//HERE  YOU CAN WRITE  WHAT IS NECESSARY 
//TO SUPSEND  PROCESS..... TO INTERUPT SAFETY

IF (Step(1000, TRUE, '<#SUSPENDING COMPONENTS#>')) THEN
 	//-------------------------------------    
	//StepCompleteWhen(Station.AutomatTask.CurrentStep.Status <> eStepStatus.Running);
		
    StepCompleteWhen( CurrentStep.Duration >= T#3000MS);
    //-------------------------------------
END_IF

IF (Step(30000, TRUE, 'SUSPEND DONE')) THEN
    //-------------------------------------
		
        THIS^._done:=TRUE;
		THIS^.Task.DoneWhen(TRUE);
	
   
    //-------------------------------------	
END_IF
END_METHOD

METHOD PUBLIC OnStart
SUPER^.OnStart();
Station.RecoverTask.Restore();
END_METHOD

PROPERTY Station : REFERENCE TO CU00x
GET
VAR
    _station : POINTER TO CU00x;
END_VAR
IF __QUERYPOINTER(Parent, _station) THEN // Check if _Parent is Station001
    Station REF= _station^;              // If the check is successful dereference a pointer. simlar to THIS^ or SUPER^
END_IF
END_GET
END_PROPERTY

END_FUNCTION_BLOCK

// ---- Abstractions/CUBase/Tasks/CUBaseSuspend.TcPOU
FUNCTION_BLOCK ABSTRACT CUBaseSuspend EXTENDS TcoTaskedSequencer
VAR
	_done:BOOL;

END_VAR

PROPERTY Done : bool
GET
Done := _done;
END_GET
END_PROPERTY

METHOD PUBLIC OnStart
_done:=FALSE;
END_METHOD

PROPERTY StationBase : REFERENCE TO CuBase
GET
VAR
    _station : POINTER TO CuBase;
END_VAR
IF __QUERYPOINTER(Parent, _station) THEN // Check if _Parent is Station001
    StationBase REF= _station^;              // If the check is successful dereference a pointer. simlar to THIS^ or SUPER^
END_IF
END_GET
END_PROPERTY

END_FUNCTION_BLOCK

// ---- Technology/CU00x/Safety/Recover/CU00xRecoverTask.TcPOU
FUNCTION_BLOCK CU00xRecoverTask EXTENDS CUBaseRecover IMPLEMENTS ICUTask
VAR
	_sb : TcoCore.StringBuilder;
END_VAR

Run();

(*~
	<docu>
		<summary>
			Main method of the sequener. Custom code needs to be placed here. The sequencer is executed by call of **Instance.Run()** method.
			This method is abstract, and it must be overridden in derived block.
		</summary>
	</docu>
~*)
METHOD PROTECTED Main : BOOL
(*

	RECOVER PROCESS 
	Following steps provide recover action for this controlled unit.
	Add components add write customized sequence according to your need.
*)

		
//
IF (Step(100, TRUE, '<#WAITING FOR START#>')) THEN
    //-------------------------------------    

    StepCompleteWhen(TRUE);
    //-------------------------------------
END_IF

//HERE  YOU CAN WRITE  WHAT IS NECESSARY 
//TO RECOVER AFTER INTERUPTED PROCESS.....

IF (Step(1000, TRUE, '<#RECOVER ANY COMPONENTS#>')) THEN
    //-------------------------------------    

    StepCompleteWhen(CurrentStep.Duration >= T#3000MS);
    //-------------------------------------
END_IF

IF (Step(30000, TRUE, 'RECOVER DONE')) THEN
    //-------------------------------------
		
        this^._done:=true;
		THIS^.Task.DoneWhen(TRUE);
		
   
    //-------------------------------------	
END_IF
END_METHOD

METHOD PUBLIC OnStart
SUPER^.OnStart();
Station.SuspendTask.Restore();
END_METHOD

PROPERTY Station : REFERENCE TO CU00x
GET
VAR
    _station : POINTER TO CU00x;
END_VAR
IF __QUERYPOINTER(Parent, _station) THEN // Check if _Parent is Station001
    Station REF= _station^;              // If the check is successful dereference a pointer. simlar to THIS^ or SUPER^
END_IF
END_GET
END_PROPERTY

END_FUNCTION_BLOCK

// ---- Abstractions/CUBase/Tasks/CUBaseRecover.TcPOU
FUNCTION_BLOCK ABSTRACT CUBaseRecover EXTENDS TcoTaskedSequencer
VAR
	_done:BOOL;

END_VAR

PROPERTY Done : bool
GET
Done := _done;
END_GET
END_PROPERTY

METHOD PUBLIC OnStart
_done:=FALSE;
END_METHOD

PROPERTY StationBase : REFERENCE TO CuBase
GET
VAR
    _station : POINTER TO CuBase;
END_VAR
IF __QUERYPOINTER(Parent, _station) THEN // Check if _Parent is Station001
    StationBase REF= _station^;              // If the check is successful dereference a pointer. simlar to THIS^ or SUPER^
END_IF
END_GET
END_PROPERTY

END_FUNCTION_BLOCK

// ---- Technology/CU00x/Positions/Cu00xTestPositions.TcPOU
FUNCTION_BLOCK Cu00xTestPositions EXTENDS TcoDrivesBeckhoff.TcoSingleAxisPositionsRootContainer
VAR_INPUT
END_VAR
VAR_OUTPUT
END_VAR
VAR
	{attribute addProperty Name "<#Pick Position#>"}
	PickPosition:TcoDrivesBeckhoff.TcoSingleAxisMoveParam;
	{attribute addProperty Name "<#Place  Position#>"}
	PlacePosition:TcoDrivesBeckhoff.TcoSingleAxisMoveParam;
END_VAR

END_FUNCTION_BLOCK

// ---- Technology/CU00x/Positions/CU00xTestMultiPositions.TcPOU
FUNCTION_BLOCK CU00xTestMultiPositions EXTENDS TcoDrivesBeckhoff.TcoMultiAxisPositionsRootContainer
VAR_INPUT
END_VAR
VAR_OUTPUT
END_VAR
VAR
	{attribute addProperty Name "<#Pick Position#>"}
	PickPosition:TcoDrivesBeckhoff.TcoMultiAxisMoveParam;
	{attribute addProperty Name "<#Place  Position#>"}
	PlacePosition:TcoDrivesBeckhoff.TcoMultiAxisMoveParam;

END_VAR

PROPERTY PUBLIC PickPos : REFERENCE TO TcoDrivesBeckhoff.TcoMultiAxisMoveParam;
GET
PickPos REF=PickPosition;
END_GET
END_PROPERTY

PROPERTY PUBLIC PlacePos : REFERENCE TO TcoDrivesBeckhoff.TcoMultiAxisMoveParam;
GET
PlacePos REF=PlacePosition;
END_GET
END_PROPERTY

END_FUNCTION_BLOCK

// ---- Abstractions/Generic/LightTower/TcoLightTower.TcPOU
FUNCTION_BLOCK TcoLightTower EXTENDS TcoCore.TcoComponent
VAR_IN_OUT
	{attribute clr [RenderIgnore()]}
	inoGreenLight   :  BOOL;
	
	{attribute clr [RenderIgnore()]}
	inoRedLight     :  BOOL;
	
	{attribute clr [RenderIgnore()]}
	inoOrangeLight  :  BOOL;
	
	{attribute clr [RenderIgnore()]}
	inoBlueLight    :  BOOL;

	{attribute clr [RenderIgnore()]}
	inoHorn         :  BOOL;
END_VAR

VAR
	
	
	{attribute addProperty Name "<#Status#>"}
    {attribute clr [ReadOnly()]}
    _status : TcoLightTower_Status;

	{attribute addProperty Name "<#Config#>"}
    _config : TcoLightTower_Config;
	
    _materrialError : bool;

	{attribute clr [RenderIgnore()]}
	_controlledUnits      : ARRAY [0..12] OF ICUBase;
				
	
	
	// group states

	{attribute clr [RenderIgnore()]}
	_blinker              : TcoUtilities.TcoBlinker(THIS^);
	{attribute clr [RenderIgnore()]}
	_blinkerSlow              : TcoUtilities.TcoBlinker(THIS^);
	

END_VAR

IF _controlledUnits[0] = 0 THEN
    THIS^.Messenger.Programming('<#Missing link to Controlled unit! No function is being executed!#>');
    RETURN;
END_IF

inoGreenLight := FALSE;
inoRedLight := FALSE;
inoOrangeLight := FALSE;
inoBlueLight := FALSE;
inoHorn := FALSE;

_blinker(inOffTime := T#500MS, inOnTime := T#500MS); //2 Hz
_blinkerSlow(inOffTime := T#1250MS, inOnTime := T#1250MS); //0.8 Hz

THIS^.Initialize();

//ground
IF _status.State.AnyGrounding THEN
    inoGreenLight := _blinker.IsOn;
    inoRedLight := _status.State.AnyInError AND _blinker.IsOn;
    inoOrangeLight := _status.State.AnyInWarning AND _blinker.IsOn;
END_IF

//auto
IF _status.State.AllInAuto AND NOT _status.State.AnyInStepMode AND NOT _status.State.AnyInError AND _status.State.AnyInWarning THEN
    inoGreenLight := TRUE; // ok production
ELSIF _status.State.AllInAuto AND _status.State.AnyInStepMode THEN
    inoGreenLight := _blinker.IsOn; //step mode
ELSIF _status.State.AllInAuto AND NOT _status.State.AnyInStepMode THEN
    inoGreenLight := TRUE; // ok production
    inoRedLight := _status.State.AnyInError AND _blinker.IsOn;
    inoOrangeLight := _status.State.AnyInWarning AND _blinker.IsOn;
ELSIF _status.State.AllInManual  THEN

    inoOrangeLight :=  _blinker.IsOn;

END_IF;

IF NOT _config.HornEnabled THEN
    inoHorn := FALSE;
END_IF;

//todo blue should be suitable for material feeding
IF _materrialError AND _status.State.AllInAuto THEN
	inoBlueLight :=  _blinker.IsOn;
END_IF

METHOD AddControlledUnit : BOOL
VAR_INPUT
 	inControlledUnit : ICUBase;
END_VAR
VAR
	i : UINT;
END_VAR
AddControlledUnit := FALSE;

IF inControlledUnit = 0 THEN
	RETURN;
END_IF

FOR i := 0 TO _config.MaxControledUnits DO
	IF _controlledUnits[i] = inControlledUnit THEN
		AddControlledUnit := TRUE;
		RETURN;
	END_IF
	
	IF 	_controlledUnits[i] = 0 THEN
		_controlledUnits[i] := inControlledUnit;
		AddControlledUnit    := TRUE;
		RETURN;
	END_IF
END_FOR
END_METHOD

PROPERTY Config :REFERENCE TO TcoLightTower_Config
GET
Config ref=_config;
END_GET
END_PROPERTY

METHOD Initialize : BOOL
VAR
	i : UINT;

END_VAR
_status.State.AllInAuto := TRUE;
_status.State.AllInGrounding := TRUE;
_status.State.AllInManual := TRUE;
_status.State.AllIdle := TRUE;
_status.State.AllGrounded := TRUE;
_status.State.AllInStepMode := TRUE;
_status.State.AllSuspended := TRUE;
_status.State.AllRecovered := TRUE;
_status.State.AllInactiveOrManualOrGrounded :=true;
_status.State.AnyInAuto := FALSE;
_status.State.AnyInManual := FALSE;
_status.State.AnyGrounding := FALSE;
_status.State.AnyInStepMode := FALSE;

_status.State.AnyInWarning := FALSE;
_status.State.AnyInError := FALSE;

i := 0;

FOR i := 0 TO _config.MaxControledUnits DO
    IF _controlledUnits[i] <> 0 THEN
        _status.State.AllInAuto := _status.State.AllInAuto AND _controlledUnits[i].StatusInfo.Mode = eCUMode.AutomatMode;
        _status.State.AllInManual := _status.State.AllInManual AND _controlledUnits[i].StatusInfo.Mode = eCUMode.ManualMode;
        _status.State.AllIdle := _status.State.AllIdle AND _controlledUnits[i].StatusInfo.Mode = eCUMode.NoMode;
        _status.State.AllInGrounding := _status.State.AllInGrounding AND
            (_controlledUnits[i].StatusInfo.Mode = eCUMode.GroundModeDone XOR
            _controlledUnits[i].StatusInfo.Mode = eCUMode.GroundMode);
        _status.State.AllGrounded := _status.State.AllGrounded AND _controlledUnits[i].StatusInfo.Mode = eCUMode.GroundModeDone;
        _status.State.AllInStepMode := _status.State.AllInStepMode AND _controlledUnits[i].StatusInfo.CurrentIsInStepMode;
        _status.State.AllSuspended := _status.State.AllSuspended AND _controlledUnits[i].SuspendTask.Task.Done;
		_status.State.AllRecovered := _status.State.AllRecovered AND _controlledUnits[i].RecoverTask.Task.Done;
		_status.State.AllInactiveOrManualOrGrounded := _status.State.AllInactiveOrManualOrGrounded 
											AND (_controlledUnits[i].StatusInfo.Mode = eCUMode.ManualMode 
												OR _controlledUnits[i].StatusInfo.Mode = eCUMode.NoMode 
												OR _controlledUnits[i].StatusInfo.Mode = eCUMode.GroundModeDone );
		
        _status.State.AnyInAuto := _status.State.AnyInAuto OR _controlledUnits[i].StatusInfo.Mode = eCUMode.AutomatMode;
        _status.State.AnyInManual := _status.State.AnyInManual OR _controlledUnits[i].StatusInfo.Mode = eCUMode.ManualMode;
        _status.State.AnyInStepMode := _status.State.AnyInStepMode OR _controlledUnits[i].StatusInfo.CurrentIsInStepMode;
        _status.State.AnyGrounding := _status.State.AnyGrounding OR
            (_controlledUnits[i].StatusInfo.Mode = eCUMode.GroundModeDone OR
            _controlledUnits[i].StatusInfo.Mode = eCUMode.GroundMode);
		_status.State.AnyInWarning := _status.State.AnyInWarning OR _controlledUnits[i].StatusInfo.State =eCUState.HasWarning;	
		_status.State.AnyInError := _status.State.AnyInError  OR _controlledUnits[i].StatusInfo.State =eCUState.HasError;	
	

    ELSE
        EXIT;
    END_IF
END_FOR
END_METHOD

PROPERTY PUBLIC MaterialError : Reference to BOOL
GET
MaterialError ref=_materrialError;
END_GET
END_PROPERTY

METHOD Restore :  TcoCore.ITcoRestorable
VAR
	i : UINT;
END_VAR
// clear all linked Controlled units
FOR i := 0 TO _config.MaxControledUnits DO
	_controlledUnits[i] := 0;
END_FOR



THIS^.Messenger.UnPin();
END_METHOD

(*~
	<docu>
		<summary>
		    Custom service (manual, maintenance) logic.
			This method must be implemented in derived class.
		</summary>			
	</docu>	
~*)
METHOD PROTECTED  ServiceMode
END_METHOD

PROPERTY Status : REFERENCE TO TcoLightTower_Status
GET
Status REF=_status;
END_GET
END_PROPERTY

END_FUNCTION_BLOCK

// ---- Abstractions/Safety/ControlButtons/TcoControlButtons.TcPOU
{attribute wpf [Container(Layout.Stack)]}
{attribute wpf [Group(Layout.GroupBox)]}

FUNCTION_BLOCK TcoControlButtons EXTENDS TcoCore.TcoObject IMPLEMENTS ITcoControlButtons
VAR_INPUT
    {attribute clr [RenderIgnore()]}
    refButtonRecover : REFERENCE TO BOOL;
    {attribute clr [RenderIgnore()]}
    refButtonSuspend : REFERENCE TO BOOL;
	{attribute clr [RenderIgnore()]}
    refButtonGround : REFERENCE TO BOOL;
    {attribute clr [RenderIgnore()]}
    refButtonAuto : REFERENCE TO BOOL;
    {attribute clr [RenderIgnore()]}
    refButtonRecoverLight : REFERENCE TO BOOL;
    {attribute clr [RenderIgnore()]}
    refButtonSuspendLight : REFERENCE TO BOOL;
    {attribute clr [RenderIgnore()]}
    refButtonGroundLight : REFERENCE TO BOOL;
    {attribute clr [RenderIgnore()]}
    refButtonAutoLight : REFERENCE TO BOOL;

END_VAR
VAR


    {attribute addProperty Name "<#ButtonRecover#>"}
    _buttonRecover : TcoElements.TcoDi(THIS^);

    {attribute addProperty Name "<#ButtonSuspend#>"}
    _buttonSuspend : TcoElements.TcoDi(THIS^);

    {attribute addProperty Name "<#ButtonGround#>"}
    _buttonGround : TcoElements.TcoDi(THIS^);

    {attribute addProperty Name "<#ButtonAuto#>"}
    _buttonAuto : TcoElements.TcoDi(THIS^);



    {attribute addProperty Name "<#ButtonRecoverLight#>"}
    _buttonRecoverLight : TcoElements.TcoDo(THIS^);

    {attribute addProperty Name "<#ButtonSuspendLight#>"}
    _buttonSuspendLight : TcoElements.TcoDo(THIS^);

    {attribute addProperty Name "<#ButtonGroundLight#>"}
    _buttonGroundLight : TcoElements.TcoDo(THIS^);
    {attribute addProperty Name "<#ButtonAutoLight#>"}
    _buttonAutoLight : TcoElements.TcoDo(THIS^);



END_VAR

IF __ISVALIDREF(refButtonRecover) THEN
    _buttonRecover(inoSignal := refButtonRecover);
END_IF

IF __ISVALIDREF(refButtonSuspend) THEN
    _buttonSuspend(inoSignal := refButtonSuspend);
END_IF;

IF __ISVALIDREF(refButtonGround) THEN
    _buttonGround(inoSignal := refButtonGround);
END_IF;

IF __ISVALIDREF(refButtonAuto) THEN
    _buttonAuto(inoSignal := refButtonAuto);
END_IF;

IF __ISVALIDREF(refButtonGroundLight) THEN
    _buttonGroundLight(inoSignal := refButtonGroundLight);
END_IF

IF __ISVALIDREF(refButtonSuspendLight) THEN
    _buttonSuspendLight(inoSignal := refButtonSuspendLight);

END_IF;

IF __ISVALIDREF(refButtonRecoverLight) THEN
    _buttonRecoverLight(inoSignal := refButtonRecoverLight);

END_IF;

IF __ISVALIDREF(refButtonAutoLight) THEN
    _buttonAutoLight(inoSignal := refButtonAutoLight);

END_IF;

PROPERTY ButtonAuto : BOOL
GET
ButtonAuto :=  _buttonAuto._signal;
END_GET
SET
// Light up illumination of button
IF ButtonAuto THEN
	_buttonAutoLight.Set();
ELSE
	_buttonAutoLight.Reset();
END_IF
END_SET
END_PROPERTY

PROPERTY ButtonGround : BOOL
GET
ButtonGround :=  _buttonGround._signal;
END_GET
SET
// Light up illumination of button
IF ButtonGround THEN
	_buttonGroundLight.Set();
ELSE
	_buttonGroundLight.Reset();
END_IF
END_SET
END_PROPERTY

PROPERTY ButtonRecover : BOOL
GET
ButtonRecover := _buttonRecover._signal;
END_GET
SET
// Light up illumination of button
IF ButtonRecover THEN
	_buttonRecoverLight.Set();
ELSE
	_buttonRecoverLight.Reset();
END_IF
END_SET
END_PROPERTY

PROPERTY ButtonSuspend : BOOL
GET
ButtonSuspend := _buttonSuspend._signal;
END_GET
SET
// Light up illumination of button
IF ButtonSuspend THEN
	_buttonSuspendLight.Set();
ELSE
	_buttonSuspendLight.Reset();
END_IF
END_SET
END_PROPERTY

(*~
	<docu>
		<summary>
			Restores this instance to the Ready state. Can be called explicitly or from within one of the restore mechanisms.	
		</summary>			
	</docu>	
~*)
METHOD  Restore : ITcoRestorable
_buttonAutoLight.Reset();
_buttonGroundLight.Reset();
_buttonSuspendLight.Reset();
_buttonRecoverLight.Reset();
END_METHOD

(*~
	<docu>
		<summary>
		    Custom service (manual, maintenance) logic.
			This method must be implemented in derived class.
		</summary>			
	</docu>	
~*)
METHOD PROTECTED  ServiceMode
THIS^._buttonRecoverLight.Service();
THIS^._buttonSuspendLight.Service();
THIS^._buttonGroundLight.Service();
THIS^._buttonAutoLight.Service();
END_METHOD

END_FUNCTION_BLOCK

// ---- Abstractions/Safety/ControlledZone/TcoControlledZone.TcPOU
FUNCTION_BLOCK TcoControlledZone EXTENDS TcoCore.TcoComponent
VAR_INPUT
    {attribute clr [RenderIgnore()]}
    inDoorCircuit : ITcoDoorCircuit;

    {attribute clr [RenderIgnore()]}
    inAirPressureOK : BOOL;

    //	{attribute clr [RenderIgnore()]}
    //	inEstopActive		      : BOOL;

END_VAR

VAR

    {attribute addProperty Name "<#Status#>"}
    {attribute clr [ReadOnly()]}
    _status : TcoControlledZone_Status;

    {attribute addProperty Name "<#Config#>"}
    _config : TcoControlledZone_Config;

    {attribute clr [RenderIgnore()]}
    _controlledUnits : ARRAY[0..12] OF ICUBase;

    {attribute clr [RenderIgnore()]}
    _controlButtons : ARRAY[0..4] OF ITcoControlButtons;

    {attribute clr [RenderIgnore()]}
    _controlKeyMode : ARRAY[0..2] OF ITcoKeyMode;

    {attribute clr [RenderIgnore()]}
    _controlKeyNormalService : ARRAY[0..2] OF ITcoKeyNormalSevice;

    // group states

    {attribute clr [CompilerOmits("BuilderPlainer", "BuilderOnliner","BuilderOnlinerInterface","BuilderShadowerInterface")]}
    _blinker : TcoUtilities.TcoBlinker(THIS^);
    {attribute clr [CompilerOmits("BuilderPlainer", "BuilderOnliner","BuilderOnlinerInterface","BuilderShadowerInterface")]}
    _blinkerSlow : TcoUtilities.TcoBlinker(THIS^);

    {attribute addProperty Name "<#Ground task#>"}
    _groundTask : TcoControlledZoneActionTask(THIS^);
    {attribute addProperty Name "<#Automat task#>"}
    _autoTask : TcoControlledZoneActionTask(THIS^);

    {attribute addProperty Name "<#Recover task#>"}
    _recoverTask : TcoControlledZoneActionTask(THIS^);

    {attribute addProperty Name "<#Suspend task#>"}
    _suspendTask : TcoControlledZoneActionTask(THIS^);

    {attribute addProperty Name "<#Key Auto task#>"}
    _keyAutoTask : TcoControlledZoneActionTask(THIS^);

    {attribute addProperty Name "<#Key Manual task#>"}
    _keyManualTask : TcoControlledZoneActionTask(THIS^);

    {attribute addProperty Name "<#Key Step task#>"}
    _keyStepTask : TcoControlledZoneActionTask(THIS^);

    {attribute addProperty Name "<#Key service task#>"}
    _keyServiceTask : TcoControlledZoneActionTask(THIS^);

    {attribute clr [RenderIgnore()]}
    _timerDoorsLocked : TON;
    {attribute clr [RenderIgnore()]}
    _timerAirPressureMonitor : TON;

    {attribute clr [RenderIgnore()]}
    _serviceKeyRising : R_Trig;

    {attribute clr [RenderIgnore()]}
    _serviceKeyFalling : F_Trig;

    {attribute clr [RenderIgnore()]}
    _recoverTaskInvokeFalling : F_Trig;

    {attribute clr [RenderIgnore()]}
    _suspendTaskInvokeFalling : F_Trig;

    {attribute clr [RenderIgnore()]}
    _recoverTaskInvokeRising : R_Trig;

    {attribute clr [RenderIgnore()]}
    _suspendTaskInvokeRising : R_Trig;

    {attribute clr [RenderIgnore()]}
    _groundTaskInvokeFalling : F_Trig;

    {attribute clr [RenderIgnore()]}
    _autoTaskInvokeFalling : F_Trig;

    {attribute clr [RenderIgnore()]}
    _groundTaskInvokeRising : F_Trig;

    {attribute clr [RenderIgnore()]}
    _autoTaskInvokeRising : F_Trig;

    {attribute clr [RenderIgnore()]}
    _keyAutoTaskInvokeFalling : F_Trig;
    {attribute clr [RenderIgnore()]}
    _keyAutoTaskInvokeRising : R_Trig;

    {attribute clr [RenderIgnore()]}
    _keyManualTaskInvokeFalling : F_Trig;
    {attribute clr [RenderIgnore()]}
    _keyManualTaskInvokeRising : R_Trig;

    {attribute clr [RenderIgnore()]}
    _keyStepTaskInvokeFalling : F_Trig;
    {attribute clr [RenderIgnore()]}
    _keyStepTaskInvokeRising : R_Trig;

    {attribute clr [RenderIgnore()]}
    _keyServiceTaskInvokeFalling : F_Trig;
    {attribute clr [RenderIgnore()]}
    _keyServiceTaskInvokeRising : R_Trig;

    _airPressureOk : BOOL;
    _conditionToRunAreSufficient : BOOL;
END_VAR

IF _controlledUnits[0] = 0 THEN
    THIS^.Messenger.Programming('<#Missing link to Controlled unit! No function is being executed!#>');
    RETURN;
END_IF

IF _controlButtons[0] = 0 
	OR _controlKeyMode[0] = 0 
	OR _controlKeyNormalService[0] = 0  THEN
    THIS^.Messenger.Programming('<#Missing link to control panel components (Buttons, Mode Keys, Normal/Service)! No function is being executed!#>');
    RETURN;
END_IF



_blinker(inOffTime := T#500MS, inOnTime := T#500MS);		//2 Hz
_blinkerSlow(inOffTime := T#1250MS, inOnTime := T#1250MS);	//0.8 Hz

THIS^.Initialize();

//presure monitoring
_airPressureOk:=TRUE;
_timerAirPressureMonitor(IN:=NOT inAirPressureOK,PT:=_config.AirPressureErrorTime);
IF _timerAirPressureMonitor.Q THEN
	_airPressureOk:=FALSE;
    THIS^.Messenger.Error('<#Air pressure is not sufficient!#>').Pin();
END_IF;

//Estop monitoring
//IF THIS^.inEstopActive THEN
//    inDoorCircuit.UnLock();
//    THIS^.Messenger.Error('<#Emergency stop active: Unlocking doors!#>').Pin();
//END_IF
// Global Voltage monitoring
IF NOT inDoorCircuit.IsGlobalVoltageOk THEN
    inDoorCircuit.UnLock();
    THIS^.Messenger.Error('<#Global control voltage interrupted: Unlocking doors!#>').Pin();
END_IF

//Voltage monitoring todo
_timerDoorsLocked(IN := inDoorCircuit.IsClosed AND inDoorCircuit.IsLocked AND  inDoorCircuit.IsLocalDoorsVoltageOk, PT := _config.DoorsLocked);

IF _timerDoorsLocked.Q THEN
    IF NOT inDoorCircuit.IsLocalVoltageOk THEN
        // unlock doors in case that control voltage goes down and it shouldn't
        inDoorCircuit.UnLock();
        THIS^.Messenger.Error('<#Local voltage interrupted: Unlocking doors!#>');
    END_IF
END_IF


_conditionToRunAreSufficient:=(inAirPressureOK OR _timerAirPressureMonitor.ET<_timerAirPressureMonitor.PT) (*AND NOT inEstopActive*)  AND inDoorCircuit.IsGlobalVoltageOk AND inDoorCircuit.IsLocalVoltageOk;
 


_recoverTaskInvokeRising(CLK:=_status.State.AnyButtonRecover);
_recoverTaskInvokeFalling(CLK:=_status.State.AnyButtonRecover);
IF _recoverTaskInvokeRising.Q THEN
	_recoverTask.Restore();
END_IF
IF _recoverTaskInvokeFalling.Q THEN
	_recoverTask.Invoke();
	_suspendTask.Restore();
END_IF



_suspendTaskInvokeRising(CLK:=_status.State.AnyButtonSuspend);
_suspendTaskInvokeFalling(CLK:=_status.State.AnyButtonSuspend);
IF _suspendTaskInvokeRising.Q THEN
	_suspendTask.Restore();
END_IF
IF _suspendTaskInvokeFalling.Q THEN
	_suspendTask.Invoke();
	_recoverTask.Restore();
END_IF





_groundTaskInvokeRising(CLK:=_status.State.AnyButtonGround);
IF _groundTaskInvokeRising.Q THEN
	_groundTask.Restore();
END_IF
_groundTaskInvokeFalling(CLK:=_status.State.AnyButtonGround);
IF _groundTaskInvokeFalling.Q THEN
	_groundTask.Invoke();
END_IF
_groundTask.Enabled:= (_conditionToRunAreSufficient
						AND inDoorCircuit.IsLocalDoorsVoltageOk 
						AND _status.State.AllKeysAuto 
						AND _status.State.AllKeysNormal) ;

IF _groundTask.Busy THEN
	_autoTask.Restore();
END_IF						
						
_autoTaskInvokeRising(CLK:=_status.State.AnyButtonAuto);
IF _autoTaskInvokeRising.Q THEN
	_autoTask.Restore();
END_IF

_autoTaskInvokeFalling(CLK:=_status.State.AnyButtonAuto);
IF _autoTaskInvokeFalling.Q THEN
	_autoTask.Invoke();
END_IF

_autoTask.Enabled:= (_conditionToRunAreSufficient 
					AND inDoorCircuit.IsLocalDoorsVoltageOk 
					AND _status.State.AllKeysAuto 
					AND _status.State.AllKeysNormal) ;





//----------keys -----------

// key auto
_keyAutoTaskInvokeFalling(CLK:= _status.State.AllKeysAuto);
_keyAutoTaskInvokeRising(CLK:=_status.State.AllKeysAuto);

IF _keyAutoTaskInvokeRising.Q THEN
	_keyAutoTask.Invoke();
END_IF
IF _keyAutoTaskInvokeFalling.Q THEN
	_keyAutoTask.Restore();
END_IF


// key manual
_keyManualTaskInvokeRising(CLK:= _status.State.AnyKeyManual);
_keyManualTaskInvokeFalling(CLK:=_status.State.AnyKeyManual);

IF _keyManualTaskInvokeRising.Q THEN
	_keyManualTask.Invoke();
END_IF
IF _keyManualTaskInvokeFalling.Q THEN
	_keyManualTask.Restore();
END_IF


IF _status.State.AnyKeyStep AND _keyStepTask.Ready THEN
	_keyStepTask.Invoke();
END_IF
IF _status.State.AnyKeyStep AND _keyStepTask.Done THEN
	_keyStepTask.Restore();
END_IF

_keyStepTaskInvokeFalling(CLK:=_status.State.AnyKeyStep);

IF _keyStepTaskInvokeFalling.Q THEN
	_keyStepTask.Restore();
END_IF


// key service
_keyServiceTaskInvokeRising(CLK:= _status.State.AnyKeyService);
_keyServiceTaskInvokeFalling(CLK:=_status.State.AnyKeyService);

IF _keyServiceTaskInvokeRising.Q THEN
	_keyServiceTask.Invoke();
END_IF
IF _keyServiceTaskInvokeFalling.Q THEN
	_keyServiceTask.Restore();
END_IF






// Handling of buttons
THIS^.ButtonRecover();
THIS^.ButtonSuspend();
THIS^.ButtonGround();
THIS^.ButtonAuto();


// Handling of key 1
THIS^.KeyAuto();
THIS^.KeyManual();
THIS^.KeyStep();

// Handling of Key Normal/Service
THIS^.KeyService();

METHOD AddControlButtons : BOOL
VAR_INPUT
 	inControlButtons : ITcoControlButtons;
END_VAR
VAR
	i : UINT;
END_VAR
AddControlButtons := FALSE;

IF inControlButtons = 0 THEN
	RETURN;
END_IF

FOR i := 0 TO _config.MaxControlButtons DO
	IF _controlButtons[i] = inControlButtons THEN
		AddControlButtons := TRUE;
		RETURN;
	END_IF
	
	IF 	_controlButtons[i] = 0 THEN
		_controlButtons[i] := inControlButtons;
		AddControlButtons  := TRUE;
		RETURN;
	END_IF
END_FOR
END_METHOD

METHOD AddControlledUnit : BOOL
VAR_INPUT
 	inControlledUnit : ICUBase;
END_VAR
VAR
	i : UINT;
END_VAR
AddControlledUnit := FALSE;

IF inControlledUnit = 0 THEN
	RETURN;
END_IF

FOR i := 0 TO _config.MaxControledUnits DO
	IF _controlledUnits[i] = inControlledUnit THEN
		AddControlledUnit := TRUE;
		RETURN;
	END_IF
	
	IF 	_controlledUnits[i] = 0 THEN
		_controlledUnits[i] := inControlledUnit;
		AddControlledUnit    := TRUE;
		RETURN;
	END_IF
END_FOR
END_METHOD

METHOD AddKeyMode : BOOL
VAR_INPUT
 	inKeyMode : ITcoKeyMode;
END_VAR
VAR
	i : UINT;
END_VAR
AddKeyMode := FALSE;

IF inKeyMode = 0 THEN
	RETURN;
END_IF

FOR i := 0 TO  _config.MaxKeyMode DO
	IF _controlKeyMode[i] = inKeyMode THEN
		AddKeyMode := TRUE;
		RETURN;
	END_IF
	
	IF 	_controlKeyMode[i] = 0 THEN
		_controlKeyMode[i] := inKeyMode;
		AddKeyMode    := TRUE;
		RETURN;
	END_IF
END_FOR
END_METHOD

METHOD AddKeyNormalService : BOOL
VAR_INPUT
 	inKeyNormalService : ITcoKeyNormalSevice;
END_VAR
VAR
	i : UINT;
END_VAR
AddKeyNormalService := FALSE;

IF inKeyNormalService = 0 THEN
	RETURN;
END_IF

FOR i := 0 TO _config.MaxKeyNormalService DO
	IF _controlKeyNormalService[i] = inKeyNormalService THEN
		AddKeyNormalService := TRUE;
		RETURN;
	END_IF
	
	IF 	_controlKeyNormalService[i] = 0 THEN
		_controlKeyNormalService[i] := inKeyNormalService;
		AddKeyNormalService    := TRUE;
		RETURN;
	END_IF
END_FOR
END_METHOD

PROPERTY PUBLIC AirPressureOk : bool
GET
AirPressureOk:=_airPressureOk;
END_GET
END_PROPERTY

{attribute 'monitoring' := 'variable'}
PROPERTY AnyButtonAuto : BOOL
GET
AnyButtonAuto := _status.State.AnyButtonAuto;
END_GET
SET
VAR
	button : UINT;
END_VAR
FOR button := 0 TO _config.MaxControlButtons DO
	IF _controlButtons[button] <> 0 THEN
		_controlButtons[button].ButtonAuto := AnyButtonAuto;
	ELSE
		EXIT;
	END_IF
END_FOR
END_SET
END_PROPERTY

{attribute 'monitoring' := 'variable'}
PROPERTY AnyButtonGround : BOOL
GET
AnyButtonGround := _Status.State.AnyButtonGround;
END_GET
SET
VAR
	button : UINT;
END_VAR
FOR button := 0 TO _config.MaxControlButtons DO
	IF _controlButtons[button] <> 0 THEN
		_controlButtons[button].ButtonGround := AnyButtonGround;
	ELSE
		EXIT;
	END_IF
END_FOR
END_SET
END_PROPERTY

{attribute 'monitoring' := 'variable'}
PROPERTY AnyButtonRecover : BOOL
GET
AnyButtonRecover := _status.State.AnyButtonRecover;
END_GET
SET
VAR
	button : UINT;
END_VAR
FOR button := 0 TO _config.MaxControlButtons DO
	IF _controlButtons[button] <> 0 THEN
		_controlButtons[button].ButtonRecover := AnyButtonRecover;
	ELSE
		EXIT;
	END_IF
END_FOR
END_SET
END_PROPERTY

{attribute 'monitoring' := 'variable'}
PROPERTY AnyButtonSuspend : BOOL
GET
AnyButtonSuspend := _status.State.AnyButtonSuspend;
END_GET
SET
VAR
	button : UINT;
END_VAR
FOR button := 0 TO _config.MaxControlButtons DO
	IF _controlButtons[button] <> 0 THEN
		_controlButtons[button].ButtonSuspend := AnyButtonSuspend;
	ELSE
		EXIT;
	END_IF
END_FOR
END_SET
END_PROPERTY

METHOD ButtonAuto : BOOL
VAR
	cu : UINT;
END_VAR


IF _autoTask.Execute() THEN
	AnyButtonGround:=FALSE;
	AnyButtonAuto:=_blinkerSlow.IsOn ;		

	IF _autoTask.Progress =0 THEN
	
		IF 	_status.State.AllKeysAuto AND _status.State.AllKeysNormal  THEN
	
			_status.ActionDescription:= '<#Automat mode has been invoked.#>';
			FOR cu := 0 TO _config.MaxControledUnits DO
				IF _controlledUnits[cu] <> 0 THEN
					IF   _controlledUnits[cu].StatusInfo.Mode = eCUMode.GroundModeDone    THEN
						_controlledUnits[cu].AutomatTask.Task.Invoke();
					END_IF	
	
					IF _controlledUnits[cu].StatusInfo.Mode=eCUMode.AutomatMode THEN
							_controlledUnits[cu].AutomatTask.ModeController.Mode:=eSequencerMode.CyclicMode;	
					End_if;	
				ELSE
					EXIT;
				END_IF
			END_FOR
			_autoTask.Progress := _autoTask.Progress + 1;	
			RETURN;
		ELSE
			_status.ActionDescription:= '<#Mode keys are not in correct position.#>';
		END_IF;
			
	ELSE
		
		_autoTask.DoneWhen(_status.State.AllInAuto AND NOT _status.State.AnyButtonAuto);	
		 IF _autoTask.Done THEN
			 
		 	_status.ActionDescription:= '<#Automat mode has been done.#>';
			AnyButtonAuto:=TRUE;
		END_IF;	
	END_IF;
	
	IF _status.ActionDescription<>'' THEN
		THIS^._autoTask.Messenger.Notify(_status.ActionDescription);
	END_IF;
END_IF;
END_METHOD

METHOD ButtonGround : BOOL
VAR
	cu : UINT;
END_VAR

IF _groundTask.Execute() THEN
	// led signalisation
	AnyButtonAuto:=FALSE;
	AnyButtonGround:=_blinkerSlow.IsOn ;	

	IF _groundTask.Progress =0 THEN
		IF 	_status.State.AllKeysAuto AND _status.State.AllKeysNormal  THEN
	
			_status.ActionDescription:= '<#Grounding mode has been invoked.#>';
			FOR cu := 0 TO _config.MaxControledUnits DO
				IF _controlledUnits[cu] <> 0 THEN
					IF  _controlledUnits[cu].StatusInfo.Mode<> eCUMode.GroundMode OR _controlledUnits[cu].StatusInfo.Mode<> eCUMode.GroundModeDone THEN
						_controlledUnits[cu].GroundTask.Task.Invoke();
					END_IF	
					IF _controlledUnits[cu].StatusInfo.Mode=eCUMode.GroundMode THEN
							_controlledUnits[cu].GroundTask.ModeController.Mode:=eSequencerMode.CyclicMode;	
					End_if;			
				ELSE
					EXIT;
				END_IF
			END_FOR
			
			_groundTask.Progress := _groundTask.Progress + 1;	
			RETURN;
		ELSE
			_status.ActionDescription:= '<#Mode keys are not in correct position.#>';
		END_IF;
		
	ELSE
		
		_groundTask.DoneWhen(_status.State.AllGrounded AND NOT _status.State.AnyButtonGround );	
		 IF _groundTask.Done THEN
			 _status.ActionDescription:= '<#Grounding mode has been done.#>';
			AnyButtonGround:=TRUE;
		END_IF;	
	END_IF	
	IF _status.ActionDescription<>'' THEN
		THIS^._groundTask.Messenger.Notify(_status.ActionDescription);
	END_IF;
	

END_IF;
END_METHOD

METHOD ButtonRecover : BOOL
VAR
	cu : UINT;
END_VAR

IF _recoverTask.Execute() THEN
    AnyButtonSuspend := FALSE;

    IF _recoverTask.Progress = 2 THEN
        AnyButtonRecover := _blinker.IsOn;
    ELSE
        AnyButtonRecover := _blinkerSlow.IsOn;
    END_IF;

    IF _recoverTask.Progress = 0 THEN
        FOR cu := 0 TO _config.MaxControledUnits DO
            IF _controlledUnits[cu] <> 0 THEN
                _controlledUnits[cu].RecoverTask.Restore();
            ELSE
                EXIT;
            END_IF
        END_FOR

        _status.ActionDescription := '<#Waiting to release recover button#>';
        IF NOT _status.State.AnyButtonRecover THEN
            _recoverTask.Progress := _recoverTask.Progress + 1;
            RETURN;
        END_IF;

    END_IF

    IF _recoverTask.Progress = 1 THEN
        _status.ActionDescription := '<#Check general condition to recover zone (ControlVoltage, EStops, Presure...)!#>';

        IF inDoorCircuit.IsGlobalVoltageOk AND inDoorCircuit.IsLocalVoltageOk AND inAirPressureOK
        //			AND NOT inEstopActive 
            THEN
            _recoverTask.Progress := _recoverTask.Progress + 1;

        END_IF;

    END_IF

    IF _recoverTask.Progress = 2 THEN
        _status.ActionDescription := '<#Waiting to close and lock  all doors!#>';

        THIS^.inDoorCircuit.Lock();

        IF inDoorCircuit.IsLocked AND inDoorCircuit.IsLocked AND inDoorCircuit.IsLocalDoorsVoltageOk THEN
            _recoverTask.Progress := _recoverTask.Progress + 1;

        END_IF;

    END_IF

    IF _recoverTask.Progress = 3 THEN

        _status.ActionDescription := '<#Invoke restore sequences on each stations.#>';

        IF _status.State.AllInManual OR _status.State.AllInactiveOrManualOrGrounded THEN
            _recoverTask.Progress := 100;
            RETURN;
        END_IF

        FOR cu := 0 TO _config.MaxControledUnits DO
            IF _controlledUnits[cu] <> 0 THEN
                _controlledUnits[cu].AutomatTask.SuspendStepExecution := TRUE;
                _controlledUnits[cu].RecoverTask.ModeController.Mode := eSequencerMode.CyclicMode;
                _controlledUnits[cu].RecoverTask.Task.Invoke();

            ELSE
                EXIT;
            END_IF
        END_FOR

        IF _status.State.AllRecovered THEN
            FOR cu := 0 TO _config.MaxControledUnits DO
                IF _controlledUnits[cu] <> 0 THEN
                    _controlledUnits[cu].AutomatTask.SuspendStepExecution := FALSE;
                ELSE
                    EXIT;
                END_IF
            END_FOR

            _recoverTask.Progress := _recoverTask.Progress + 1;
        END_IF

    END_IF

    IF _recoverTask.Progress = 4 THEN

        _status.ActionDescription := '<#Setup Cyclic or Step mode. It depends on key position#>';

        FOR cu := 0 TO _config.MaxControledUnits DO
            IF _controlledUnits[cu] <> 0 THEN
                IF _status.State.AllKeysAuto THEN
                    IF _controlledUnits[cu].StatusInfo.Mode = eCUMode.AutomatMode THEN
                        _controlledUnits[cu].AutomatTask.ModeController.Mode := eSequencerMode.CyclicMode;
                    ELSIF _controlledUnits[cu].StatusInfo.Mode = eCUMode.GroundMode THEN
                        _controlledUnits[cu].GroundTask.ModeController.Mode := eSequencerMode.CyclicMode;
                    END_IF
                ELSE
                    IF _controlledUnits[cu].StatusInfo.Mode = eCUMode.AutomatMode THEN
                        _controlledUnits[cu].AutomatTask.ModeController.Mode := eSequencerMode.StepMode;
                    ELSIF _controlledUnits[cu].StatusInfo.Mode = eCUMode.GroundMode THEN
                        _controlledUnits[cu].GroundTask.ModeController.Mode := eSequencerMode.StepMode;
                    END_IF
                END_IF

            ELSE
                EXIT;
            END_IF
        END_FOR

        _recoverTask.Progress := 100;

    END_IF

    IF _recoverTask.Progress = 100 THEN

        _status.ActionDescription := '<#Recover task has been done.#>';
        _recoverTask.DoneWhen(TRUE);
        AnyButtonRecover := TRUE;

    END_IF;

    IF _status.ActionDescription <> '' THEN
        THIS^._recoverTask.Messenger.Notify(_status.ActionDescription);
    END_IF;

END_IF;
END_METHOD

METHOD ButtonSuspend : BOOL
VAR
	cu : UINT;
END_VAR
IF _suspendTask.Execute() THEN
	AnyButtonRecover:=FALSE;
	AnyButtonSuspend:=_blinkerSlow.IsOn ;	
	IF _suspendTask.Progress =0 THEN
		FOR cu := 0 TO _config.MaxControledUnits DO
			IF _controlledUnits[cu] <> 0 THEN
				_controlledUnits[cu].SuspendTask.Restore();

			ELSE
				EXIT;
			END_IF
		END_FOR
		_status.ActionDescription:='<#Waiting to release suspend button#>';
		IF NOT _status.State.AnyButtonSuspend THEN
				_suspendTask.Progress := _suspendTask.Progress + 1;	
				RETURN;

		END_IF;
	
	END_IF
	
	IF _suspendTask.Progress =1 THEN
		_status.ActionDescription:='<#Check general condition to suspned zone (ControlVoltage,EStops,Presure...)!#>';
		
		IF NOT inDoorCircuit.IsGlobalVoltageOk
			OR NOT inDoorCircuit.IsLocalVoltageOk
			OR NOT inAirPressureOK
//			OR inEstopActive 
			THEN
			_suspendTask.Progress := 100;
			
			THIS^.inDoorCircuit.Unlock();
		ELSE
			_suspendTask.Progress := _suspendTask.Progress + 1;	
		END_IF;
	
	END_IF
	
	IF _suspendTask.Progress =2 THEN
		
		_status.ActionDescription:= '<#Force step mode.#>';
		
		IF _status.State.AllInManual OR _status.State.AllInactiveOrManualOrGrounded THEN
			_suspendTask.Progress := 4;
			RETURN;
		END_IF
		FOR cu := 0 TO _config.MaxControledUnits DO
			IF _controlledUnits[cu] <> 0 THEN
			

				IF _controlledUnits[cu].StatusInfo.Mode=eCUMode.AutomatMode THEN
					_controlledUnits[cu].AutomatTask.ModeController.Mode:=eSequencerMode.StepMode;
				ELSIF _controlledUnits[cu].StatusInfo.Mode=eCUMode.GroundMode THEN
					_controlledUnits[cu].GroundTask.ModeController.Mode:=eSequencerMode.StepMode;
				END_IF
		
	
			ELSE
				EXIT;
			END_IF
		END_FOR


		
		IF _status.State.AllInStepMode or true THEN
			_suspendTask.Progress := _suspendTask.Progress + 1;
		END_IF;
			
	END_IF
	
	IF _suspendTask.Progress =3 THEN
		
		_status.ActionDescription:='<#Invoke suspend sequences on each stations.#>';
		
		
		FOR cu := 0 TO _config.MaxControledUnits DO
			IF _controlledUnits[cu] <> 0 THEN
				_controlledUnits[cu].SuspendTask.ModeController.Mode := eSequencerMode.CyclicMode;
				_controlledUnits[cu].SuspendTask.Task.Invoke();

			ELSE
				EXIT;
			END_IF
		END_FOR

		IF _status.State.AllSuspended THEN
			_suspendTask.Progress := _suspendTask.Progress+1;
		END_IF
		
	END_IF
	
	
	
	IF _suspendTask.Progress =4 THEN
		_status.ActionDescription:='<#Waiting to unlock  all doors!#>';
		
		THIS^.inDoorCircuit.UnLock();
		
		IF inDoorCircuit.IsUnLocked THEN
		//	_suspendTask.Progress := 100;
	
		END_IF;
	
	END_IF


	IF _suspendTask.Progress = 100 THEN
		_status.ActionDescription:= '<#Suspend task has been done.#>';
		_suspendTask.DoneWhen(TRUE);
		AnyButtonSuspend:=TRUE;
	END_IF;	


	IF _status.ActionDescription<>'' THEN
		THIS^._suspendTask.Messenger.Notify(_status.ActionDescription);
	END_IF;
	
END_IF;
END_METHOD

PROPERTY Config :REFERENCE TO TcoControlledZone_Config
GET
Config ref=_config;
END_GET
END_PROPERTY

METHOD Initialize : BOOL
VAR
	i : UINT;

END_VAR
_status.State.AllInAuto := TRUE;
_status.State.AllInGrounding := TRUE;
_status.State.AllInManual := TRUE;
_status.State.AllIdle := TRUE;
_status.State.AllGrounded := TRUE;
_status.State.AllInStepMode := TRUE;
_status.State.AllSuspended := TRUE;
_status.State.AllRecovered := TRUE;
_status.State.AllInactiveOrManualOrGrounded :=true;
_status.State.AnyInAuto := FALSE;
_status.State.AnyInManual := FALSE;
_status.State.AnyGrounding := FALSE;
_status.State.AnyInStepMode := FALSE;

i := 0;

FOR i := 0 TO _config.MaxControledUnits DO
    IF _controlledUnits[i] <> 0 THEN
        _status.State.AllInAuto := _status.State.AllInAuto AND _controlledUnits[i].StatusInfo.Mode = eCUMode.AutomatMode;
        _status.State.AllInManual := _status.State.AllInManual AND _controlledUnits[i].StatusInfo.Mode = eCUMode.ManualMode;
        _status.State.AllIdle := _status.State.AllIdle AND _controlledUnits[i].StatusInfo.Mode = eCUMode.NoMode;
        _status.State.AllInGrounding := _status.State.AllInGrounding AND
            (_controlledUnits[i].StatusInfo.Mode = eCUMode.GroundModeDone XOR
            _controlledUnits[i].StatusInfo.Mode = eCUMode.GroundMode);
        _status.State.AllGrounded := _status.State.AllGrounded AND _controlledUnits[i].StatusInfo.Mode = eCUMode.GroundModeDone;
        _status.State.AllInStepMode := _status.State.AllInStepMode AND _controlledUnits[i].StatusInfo.CurrentIsInStepMode;
        _status.State.AllSuspended := _status.State.AllSuspended AND _controlledUnits[i].SuspendTask.Task.Done;
		_status.State.AllRecovered := _status.State.AllRecovered AND _controlledUnits[i].RecoverTask.Task.Done;
		_status.State.AllInactiveOrManualOrGrounded := _status.State.AllInactiveOrManualOrGrounded 
											AND (_controlledUnits[i].StatusInfo.Mode = eCUMode.ManualMode 
												OR _controlledUnits[i].StatusInfo.Mode = eCUMode.NoMode 
												OR _controlledUnits[i].StatusInfo.Mode = eCUMode.GroundModeDone );
		
        _status.State.AnyInAuto := _status.State.AnyInAuto OR _controlledUnits[i].StatusInfo.Mode = eCUMode.AutomatMode;
        _status.State.AnyInManual := _status.State.AnyInManual OR _controlledUnits[i].StatusInfo.Mode = eCUMode.ManualMode;
        _status.State.AnyInStepMode := _status.State.AnyInStepMode OR _controlledUnits[i].StatusInfo.CurrentIsInStepMode;
        _status.State.AnyGrounding := _status.State.AnyGrounding OR
            (_controlledUnits[i].StatusInfo.Mode = eCUMode.GroundModeDone OR
            _controlledUnits[i].StatusInfo.Mode = eCUMode.GroundMode);

    ELSE
        EXIT;
    END_IF
END_FOR

// update states of buttons
_status.State.AnyButtonRecover := FALSE;
_status.State.AnyButtonSuspend := FALSE;
_status.State.AnyButtonGround := FALSE;
_status.State.AnyButtonAuto := FALSE;
i := 0;

FOR i := 0 TO _config.MaxControlButtons DO
    IF _controlButtons[i] <> 0 THEN
        _status.State.AnyButtonRecover := _status.State.AnyButtonRecover OR _controlButtons[i].ButtonRecover;
        _status.State.AnyButtonGround := _status.State.AnyButtonGround OR _controlButtons[i].ButtonGround;
        _status.State.AnyButtonAuto := _status.State.AnyButtonAuto OR _controlButtons[i].ButtonAuto;
        _status.State.AnyButtonSuspend := _status.State.AnyButtonSuspend OR _controlButtons[i].ButtonSuspend;
    ELSE
        EXIT;
    END_IF
END_FOR

// update states of keys
_status.State.AllKeysNormal := TRUE;
_status.State.AnyKeyService := FALSE;
i := 0;

FOR i := 0 TO _config.MaxKeyNormalService DO
    IF _controlKeyNormalService[i] <> 0 THEN
        _status.State.AllKeysNormal := _status.State.AllKeysNormal AND _controlKeyNormalService[i].KeyInNormal;
        _status.State.AnyKeyService := _status.State.AnyKeyService OR _controlKeyNormalService[i].KeyInService;
    ELSE
        EXIT;
    END_IF
END_FOR

// update states of keys
_status.State.AllKeysAuto := TRUE;
_status.State.AnyKeyManual := FALSE;
_status.State.AnyKeyStep := FALSE;
i := 0;

FOR i := 0 TO _config.MaxKeyMode DO
    IF _controlKeyMode[i] <> 0 THEN
        _status.State.AllKeysAuto := _status.State.AllKeysAuto AND _controlKeyMode[i].KeyInAuto;
        _status.State.AnyKeyManual := _status.State.AnyKeyManual OR _controlKeyMode[i].KeyInManual;
        _status.State.AnyKeyStep := _status.State.AnyKeyStep OR _controlKeyMode[i].KeyInStep;
    ELSE
        EXIT;
    END_IF
END_FOR
END_METHOD

METHOD KeyAuto 
VAR
	cu : UINT;
END_VAR
IF _keyAutoTask.Execute() THEN
	_status.ActionDescription:= '<#Automatic mode is not possibe to set(All keys must be in NORMAL and AUTO!)#>';
	IF 	 _status.State.AllKeysNormal  AND _status.State.AllKeysAuto THEN
		
//			_status.ActionDescription:= '<#Automatic mode is set(Step mode is disabled)!#>';
//			FOR cu := 0 TO _config.MaxControledUnits DO
//				IF _controlledUnits[cu] <> 0 THEN
//					IF _controlledUnits[cu].StatusInfo.Mode=eCUMode.AutomatMode THEN
//						_controlledUnits[cu].AutomatTask.ModeController.Mode:=eSequencerMode.CyclicMode;
//					ELSIF _controlledUnits[cu].StatusInfo.Mode=eCUMode.GroundMode THEN
//						_controlledUnits[cu].GroundTask.ModeController.Mode:=eSequencerMode.CyclicMode;
//					END_IF
//				ELSE
//					EXIT;
//				END_IF
//			END_FOR
	
		ELSE
			_status.ActionDescription:= '<#Cyclic mode is not allowed while any control key is in Service mode!#> <#Setting step mode!#>';
			FOR cu := 0 TO _config.MaxControledUnits DO
				IF _controlledUnits[cu] <> 0 THEN
						IF _controlledUnits[cu].StatusInfo.Mode=eCUMode.AutomatMode THEN
							_controlledUnits[cu].AutomatTask.ModeController.Mode:=eSequencerMode.StepMode;
						ELSIF _controlledUnits[cu].StatusInfo.Mode=eCUMode.GroundMode THEN
							_controlledUnits[cu].GroundTask.ModeController.Mode:=eSequencerMode.StepMode;
						END_IF
				ELSE
					EXIT;
				END_IF
			END_FOR	
		END_IF;
	
	


	IF  _status.State.AllInAuto THEN
		_keyAutoTask.DoneWhen(TRUE);
	END_IF;
	
	IF _status.ActionDescription<>'' THEN
		THIS^._keyAutoTask.Messenger.Notify(_status.ActionDescription);
	END_IF;	
END_IF
END_METHOD

METHOD KeyManual 
VAR
	cu : UINT;
END_VAR

IF _keyManualTask.Execute() THEN
	_status.ActionDescription:= '<#Manual mode is not possibe to set(At least one SERVICE and one MANUAL keys must be in position!)#>';
	
	IF _keyManualTask.Progress =0 THEN
		IF _status.State.AnyKeyManual AND _status.State.AnyKeyService THEN
			IF NOT _status.State.AllInManual THEN
				_keyManualTask.Progress := _keyManualTask.Progress + 1;// all to manual
			ELSE
				_keyManualTask.Progress := _keyManualTask.Progress + 2;
			END_IF
		END_IF;
	
	END_IF

	IF _keyManualTask.Progress =1 THEN
		
		_status.ActionDescription:='<#Manual mode is starting#>';
		
		FOR cu := 0 TO _config.MaxControledUnits DO
			IF _controlledUnits[cu] <> 0 THEN
				IF  _controlledUnits[cu].StatusInfo.Mode<> eCUMode.ManualMode THEN
					_controlledUnits[cu].ManualTask.Invoke();
				END_IF			
			ELSE
				EXIT;
			END_IF
		END_FOR

		IF _status.State.AllInManual THEN
			_keyManualTask.Progress := _keyManualTask.Progress + 1;
		END_IF
		
	END_IF
	
	
	IF _keyManualTask.Progress =2 THEN
		
		_status.ActionDescription:='<#Clear step mode#>';
		
		FOR cu := 0 TO _config.MaxControledUnits DO
			IF _controlledUnits[cu] <> 0 THEN
				_controlledUnits[cu].AutomatTask.ModeController.Mode := eSequencerMode.CyclicMode;
				_controlledUnits[cu].GroundTask.ModeController.Mode := eSequencerMode.CyclicMode;		
			ELSE
				EXIT;
			END_IF
		END_FOR

		IF _status.State.AllInManual THEN
			_keyManualTask.Progress := _keyManualTask.Progress + 1;
		END_IF
		
	END_IF

	IF _keyManualTask.Progress =3 THEN
		_keyManualTask.DoneWhen(TRUE);	
	END_IF

	IF _status.ActionDescription<>'' THEN
		THIS^._keyManualTask.Messenger.Notify(_status.ActionDescription);
	END_IF;
END_IF;
END_METHOD

METHOD KeyService
VAR
	cu : UINT;
END_VAR
IF _keyServiceTask.Execute() THEN
	
	IF 	_status.State.AnyKeyManual  AND _status.State.AnyKeyService  THEN
		_status.ActionDescription:='<#Manual mode is starting due service key combination (Manual / Service)#>';
		
		FOR cu := 0 TO _config.MaxControledUnits DO
			IF _controlledUnits[cu] <> 0 THEN
				IF  _controlledUnits[cu].StatusInfo.Mode<> eCUMode.ManualMode THEN
					_controlledUnits[cu].ManualTask.Invoke();
				END_IF			
			ELSE
				EXIT;
			END_IF
		END_FOR
	ELSE
		_status.ActionDescription:='<#Step mode is required because Service key position is set!#>';
		FOR cu := 0 TO _config.MaxControledUnits DO
			IF _controlledUnits[cu] <> 0 THEN
					IF _controlledUnits[cu].StatusInfo.Mode=eCUMode.AutomatMode THEN
						_controlledUnits[cu].AutomatTask.ModeController.Mode:=eSequencerMode.StepMode;
					ELSIF _controlledUnits[cu].StatusInfo.Mode=eCUMode.GroundMode THEN
						_controlledUnits[cu].GroundTask.ModeController.Mode:=eSequencerMode.StepMode;
					END_IF
			ELSE
				EXIT;
			END_IF
		END_FOR
	END_IF;
	


	IF  _status.State.AllInStepMode OR _status.State.AllInManual THEN
		_keyServiceTask.DoneWhen(TRUE);
	END_IF;
	
	IF _status.ActionDescription<>'' THEN
		THIS^._keyServiceTask.Messenger.Notify(_status.ActionDescription);
	END_IF;	
END_IF
END_METHOD

METHOD KeyStep 
VAR
	cu : UINT;
END_VAR

IF _keyStepTask.Execute() THEN
		
	_status.ActionDescription:='<#Step mode is required but mode key is not in required position!#>';

	IF _status.State.AnyKeyStep THEN
		FOR cu := 0 TO _config.MaxControledUnits DO
			IF _controlledUnits[cu] <> 0 THEN
				IF _controlledUnits[cu].StatusInfo.Mode=eCUMode.AutomatMode THEN
					_controlledUnits[cu].AutomatTask.ModeController.Mode:=eSequencerMode.StepMode;
				ELSIF _controlledUnits[cu].StatusInfo.Mode=eCUMode.GroundMode THEN
					_controlledUnits[cu].GroundTask.ModeController.Mode:=eSequencerMode.StepMode;
				END_IF
			ELSE
				EXIT;
			END_IF
		
		END_FOR
	END_IF;
	
	IF _status.State.AllInStepMode THEN
		_status.ActionDescription:='<#Step mode is set or all are inactive!#>';
		_keyStepTask.DoneWhen(TRUE);
	END_IF;
	
	IF _status.ActionDescription<>'' THEN
		THIS^._keyStepTask.Messenger.Notify(_status.ActionDescription);
	END_IF;	
END_IF;
END_METHOD

METHOD Restore :  TcoCore.ITcoRestorable
VAR
	i : UINT;
END_VAR
// clear all linked Controlled units
FOR i := 0 TO _config.MaxControledUnits DO
	_controlledUnits[i] := 0;
END_FOR

// clear all linked Control buttons
FOR i := 0 TO _config.MaxControlButtons DO
	_controlButtons[i] := 0;
END_FOR

// clear all linked service keys (N/S)
FOR i := 0 TO _config.MaxKeyNormalService DO
	_controlKeyNormalService[i] := 0;
END_FOR

// clear all linked Sequencer keys (M/S/A)
FOR i := 0 TO _config.MaxKeyMode DO
	_controlKeyMode[i] := 0;
END_FOR


THIS^.Messenger.UnPin();
END_METHOD

(*~
	<docu>
		<summary>
		    Custom service (manual, maintenance) logic.
			This method must be implemented in derived class.
		</summary>			
	</docu>	
~*)
METHOD PROTECTED  ServiceMode
END_METHOD

METHOD Signalisation
VAR_INPUT
END_VAR

AnyButtonAuto:=_blinkerSlow.IsOn  AND _autoTask.Busy;
END_METHOD

PROPERTY Status : REFERENCE TO TcoControlledZone_Status
GET
Status REF=_status;
END_GET
END_PROPERTY

END_FUNCTION_BLOCK

// ---- Abstractions/Safety/ControlledZone/TcoControlledZoneActionTask.TcPOU
FUNCTION_BLOCK PUBLIC  TcoControlledZoneActionTask EXTENDS TcoCore.TcoTask 
VAR_IN_OUT
	inoStatus:TcoControlledZone_Status;
END_VAR
VAR
    _progress : INT := 0;
    {attribute 'hide'} 
	_infoTimer :  TON;
    {attribute 'hide'} 
	_errorTimer :  TON;
    {attribute 'hide'} 
	_varInfo : __SYSTEM.VAR_INFO;
    {attribute 'hide'} 
	_sb : TcoCore.StringBuilder;

END_VAR

(*~
	<docu>
		<summary>
			Executes when task reaches the ```Done``` state .
		</summary>			
	</docu>	
~*)
METHOD PROTECTED OnDone
_progress := 0;
END_METHOD

PROPERTY PUBLIC Progress : REFERENCE TO INT
GET
Progress ref= _progress;
END_GET
END_PROPERTY

(*~
	<docu>
		<summary>
			Restores this instance to the Ready state. Can be called explicitly or from within one of the restore mechanisms.
			<para>
				See also <see cref="PlcDocu.TcoCore.TcoTask.AutoRestorable()"/>
			</para>
		</summary>			
	</docu>	
~*)
METHOD Restore : TcoCore.ITcoRestorable
SUPER^.Restore();
_progress := 0;
Messenger.UnPin();
END_METHOD

END_FUNCTION_BLOCK

// ---- Abstractions/Safety/ControlVoltage/TcoControlVoltage.TcPOU
{attribute wpf [Container(Layout.Stack)]}
FUNCTION_BLOCK TcoControlVoltage EXTENDS TcoElements.TcoDi IMPLEMENTS  ITcoControlVoltage

VAR_OUTPUT
END_VAR
VAR
END_VAR

SUPER^(inoSignal:=inoSignal);
IF NOT inoSignal THEN
	Messenger.Error('<#Voltage is Off!#>');
END_IF;

PROPERTY IsOff : BOOL
GET
IsOff:=not this^._signal;
END_GET
END_PROPERTY

PROPERTY IsOn : BOOL
GET
IsOn:=this^._signal;
END_GET
END_PROPERTY

END_FUNCTION_BLOCK

// ---- Abstractions/Safety/DoorCircuit/TcoDoorCircuit.TcPOU
FUNCTION_BLOCK TcoDoorCircuit EXTENDS TcoCore.TcoComponent IMPLEMENTS ITcoDoorCircuit
VAR_INPUT
END_VAR
VAR_OUTPUT
END_VAR
VAR
	
	{attribute addProperty Name "<#Status#>"}
    {attribute clr [ReadOnly()]}
    _status : TcoDoorCircuit_Status;

	{attribute addProperty Name "<#Config#>"}
    _config : TcoDoorCircuit_Config;

	
	{attribute clr [RenderIgnore()]}
	_doors              : ARRAY [0..12] OF ITcoDoorLock;
	
	{attribute clr [RenderIgnore()]}
	_localDoorsVoltage  : ARRAY [0..4] OF ITcoControlVoltage;
	
	{attribute clr [RenderIgnore()]}
	_localVoltage  : ARRAY [0..4] OF ITcoControlVoltage;
	
	{attribute clr [RenderIgnore()]}
	_globalVoltage : ARRAY [0..4] OF ITcoControlVoltage;
	
	
	
    {attribute addProperty Name "<#Closed#>"}
    _isClosed : BOOL;
    
    {attribute addProperty Name "<#Locked#>"}
    _isLocked : BOOL;
    
    {attribute addProperty Name "<#Unlocked#>"}
    _isUnLocked : BOOL;
    
    {attribute addProperty Name "<#Global votage#>"}
    _isGlobalVoltageOk : BOOL;
    
    {attribute addProperty Name "<#Local voltage#>"}
    _isLocalVoltageOk : BOOL;
    
	 {attribute addProperty Name "<#Local Doors#>"}
    _isLocalDoorsVoltageOk : BOOL;


END_VAR

Initialize();

METHOD AddDoors : BOOL
VAR_INPUT
	inDoor : ITcoDoorLock;
END_VAR
VAR
	i : UINT;
END_VAR
AddDoors := FALSE;
FOR i := 0 TO _config.MaxDoors DO
	IF _doors[i] = inDoor THEN
		AddDoors := TRUE;
		RETURN;
	END_IF
	
	IF _doors[i] = 0 THEN
		_doors[i] := inDoor;
		AddDoors := TRUE;
		RETURN;
	END_IF
END_FOR
END_METHOD

METHOD AddGlobalVoltage : BOOL
VAR_INPUT
 	inVoltage : ITcoControlVoltage;
END_VAR
VAR
	i : UINT;
END_VAR
AddGlobalVoltage := FALSE;

IF inVoltage = 0 THEN
	RETURN;
END_IF

FOR i := 0 TO _config.MaxGlobalVoltage DO
	IF _globalVoltage[i] = inVoltage THEN
		addGlobalVoltage := TRUE;
		RETURN;
	END_IF
	
	IF 	_globalVoltage[i] = 0 THEN
		_globalVoltage[i] := inVoltage;
		addGlobalVoltage    := TRUE;
		RETURN;
	END_IF
END_FOR
END_METHOD

METHOD AddLocalDoorsVoltage : BOOL
VAR_INPUT
 	inVoltage : ITcoControlVoltage;
END_VAR
VAR
	i : UINT;
END_VAR
AddLocalDoorsVoltage := FALSE;

IF inVoltage = 0 THEN
	RETURN;
END_IF

FOR i := 0 TO _config.MaxLocalVoltage DO
	IF _localDoorsVoltage[i] = inVoltage THEN
		AddLocalDoorsVoltage := TRUE;
		RETURN;
	END_IF
	
	IF 	_localDoorsVoltage[i] = 0 THEN
		_localDoorsVoltage[i] := inVoltage;
		AddLocalDoorsVoltage    := TRUE;
		RETURN;
	END_IF
END_FOR
END_METHOD

METHOD AddLocalVoltage : BOOL
VAR_INPUT
 	inVoltage : ITcoControlVoltage;
END_VAR
VAR
	i : UINT;
END_VAR
addLocalVoltage := FALSE;

IF inVoltage = 0 THEN
	RETURN;
END_IF

FOR i := 0 TO _config.MaxLocalVoltage DO
	IF _localVoltage[i] = inVoltage THEN
		addLocalVoltage := TRUE;
		RETURN;
	END_IF
	
	IF 	_localVoltage[i] = 0 THEN
		_localVoltage[i] := inVoltage;
		addLocalVoltage    := TRUE;
		RETURN;
	END_IF
END_FOR
END_METHOD

PROPERTY Config :REFERENCE TO TcoDoorCircuit_Config
GET
Config ref=_config;
END_GET
END_PROPERTY

METHOD Initialize : BOOL
VAR
	d       : UINT;
	gv      : UINT;
	lv      : UINT;
	ldoors      : UINT;
	setOnce : BOOL;
END_VAR
// ------------------------------------------------------------- 
// 						GLOBAL VOLTAGE
// ------------------------------------------------------------- 
_isGlobalVoltageOk := FALSE;
setOnce            := FALSE;

FOR gv := 0 TO _config.MaxGlobalVoltage DO
	IF _globalVoltage[gv] <> 0 THEN
		IF NOT setOnce THEN
			_isGlobalVoltageOk := TRUE;
			setOnce := TRUE;
		END_IF
		
		IF _globalVoltage[gv].IsOff THEN
			_isGlobalVoltageOk := FALSE;
			EXIT;
		END_IF
	ELSE
		EXIT;
	END_IF
END_FOR

// ------------------------------------------------------------- 
// 						LOCAL VOLTAGE
// ------------------------------------------------------------- 
_isLocalVoltageOk := FALSE;
setOnce           := FALSE;

FOR lv := 0 TO _config.MaxLocalVoltage DO
	IF _localVoltage[lv] <> 0 THEN
		IF NOT setOnce THEN
			_isLocalVoltageOk := TRUE;
			setOnce := TRUE;
		END_IF
		
		IF _localVoltage[lv].IsOff THEN
			_isLocalVoltageOk := false;
			EXIT;
		END_IF
	ELSE
		EXIT;
	END_IF
END_FOR

// ------------------------------------------------------------- 
// 						LOCAL DOORS VOLTAGE OK
// ------------------------------------------------------------- 
_isLocalDoorsVoltageOk := FALSE;
setOnce           := FALSE;

FOR ldoors := 0 TO _config.MaxLocalDoorsVoltage DO
	IF _localDoorsVoltage[ldoors] <> 0 THEN
		IF NOT setOnce THEN
			_isLocalDoorsVoltageOk := TRUE;
			setOnce := TRUE;
		END_IF
		
		IF _localDoorsVoltage[ldoors].IsOff THEN
			_isLocalDoorsVoltageOk := FALSE;
			EXIT;
		END_IF
	ELSE
		EXIT;
	END_IF
END_FOR

// ------------------------------------------------------------- 
// 							DOORS
// ------------------------------------------------------------- 
_isClosed      := FALSE;
_isLocked      := FALSE;
_isUnLocked    := FALSE;
setOnce        := FALSE;
FOR d := 0 TO _config.MaxDoors DO
	IF _doors[d] <> 0 THEN
		IF NOT setOnce THEN
			setOnce        := TRUE;
			_isClosed      := TRUE;
			_isLocked      := TRUE;
			_isUnLocked    := TRUE;
		END_IF

		// Return TRUE only if all doors are Closed
		_isClosed   := _isClosed AND (_doors[d].IsClosed); // OR _doors[d].Deactivate);
		// Return TRUE only if all doors are Locked
		_isLocked   := _isLocked AND (_doors[d].IsLocked); //OR _doors[d].Deactivate);
		// Return TRUE only if all doors are Unlocked
		_isUnLocked := _isUnLocked AND NOT _doors[d].IsLocked;

	ELSE
		EXIT;
	END_IF
END_FOR
END_METHOD

{attribute 'monitoring' := 'variable'}
PROPERTY IsClosed : BOOL
GET
VAR
	d : UINT;
	setOnce : BOOL;
END_VAR
IsClosed := _isClosed ;
END_GET
END_PROPERTY

{attribute 'monitoring' := 'variable'}
PROPERTY IsGlobalVoltageOk : BOOL
GET
VAR
	gv : UINT;
END_VAR
IsGlobalVoltageOk := _isGlobalVoltageOk;
END_GET
END_PROPERTY

{attribute 'monitoring' := 'variable'}
PROPERTY IsLocalDoorsVoltageOk : BOOL
GET
VAR
	lv : UINT;
END_VAR
IsLocalDoorsVoltageOk := _isLocalDoorsVoltageOk;
END_GET
END_PROPERTY

{attribute 'monitoring' := 'variable'}
PROPERTY IsLocalVoltageOk : BOOL
GET
VAR
	lv : UINT;
END_VAR
IsLocalVoltageOk := _isLocalVoltageOk;
END_GET
END_PROPERTY

{attribute 'monitoring' := 'variable'}
PROPERTY IsLocked : BOOL
GET
VAR
	d : UINT;
	setOnce : BOOL;
END_VAR
IsLocked := _isLocked ;
END_GET
END_PROPERTY

{attribute 'monitoring' := 'variable'}
PROPERTY IsUnLocked : BOOL
GET
VAR
	d : UINT;
	setOnce : BOOL;
END_VAR
IsUnLocked := _isUnLocked;
END_GET
END_PROPERTY

METHOD Lock : BOOL
VAR_INPUT
END_VAR
VAR
	d : UINT;
END_VAR
Lock := FALSE;

IF NOT IsClosed THEN
	// we can't lock doors which are not closed
	RETURN;
END_IF

FOR d := 0 TO _config.MaxDoors DO
	IF _doors[d] <> 0 THEN
			_doors[d].Lock();
	ELSE
		EXIT;
	END_IF
END_FOR

Lock := THIS^.IsLocked;
END_METHOD

METHOD RemoveAllDoors
VAR
	i : UINT;
END_VAR
FOR i := 0 TO _config.MaxDoors DO
	_doors[i] := 0;
END_FOR
END_METHOD

METHOD RemoveDoors : BOOL
VAR_INPUT
	inDoorLock : ITcoDoorLock;
END_VAR
VAR
	i : UINT;
END_VAR
RemoveDoors := FALSE;

FOR i := 0 TO _config.MaxDoors DO 
	IF _doors[i] = inDoorLock THEN
		_doors[i] := 0;
		RemoveDoors :=  TRUE;
		RETURN;
	END_IF
END_FOR
END_METHOD

(*~
	<docu>
		<summary>
			Restores this instance to the Ready state. Can be called explicitly or from within one of the restore mechanisms.	
		</summary>			
	</docu>	
~*)
METHOD  Restore : ITcoRestorable

VAR
	i : UINT;
END_VAR
RemoveAllDoors();

FOR i := 0 TO _config.MaxGlobalVoltage DO
	_globalVoltage[i] := 0;
END_FOR

FOR i := 0 TO _config.MaxLocalVoltage DO
	_localVoltage[i] := 0;
END_FOR
FOR i := 0 TO _config.MaxLocalDoorsVoltage DO
	_localDoorsVoltage[i] := 0;
END_FOR
END_METHOD

(*~
	<docu>
		<summary>
		    Custom service (manual, maintenance) logic.
			This method must be implemented in derived class.
		</summary>			
	</docu>	
~*)
METHOD PROTECTED  ServiceMode
END_METHOD

PROPERTY Status : REFERENCE TO TcoDoorCircuit_Status
GET
Status REF=_status;
END_GET
END_PROPERTY

METHOD UnLock : BOOL
VAR
	d 		: UINT;
	setOnce : BOOL;
END_VAR
UnLock := FALSE;

FOR d := 0 TO _config.MaxDoors DO
	IF _doors[d] <> 0 THEN
		_doors[d].Unlock();
	ELSE
		exit;
	END_IF
END_FOR


FOR d := 0 TO _config.MaxDoors DO
	IF _doors[d] <> 0 THEN
		IF NOT setOnce THEN
			setOnce := TRUE;
			UnLock := TRUE;
		END_IF
		
		// return TRUE only if all doors are unlocked
		UnLock := Unlock AND NOT _doors[d].IsLocked;
	ELSE
		EXIT;
	END_IF
END_FOR
END_METHOD

END_FUNCTION_BLOCK

// ---- Abstractions/Safety/Doors/TcoStandardDoor.TcPOU
FUNCTION_BLOCK TcoStandardDoor EXTENDS TcoCore.TcoComponent IMPLEMENTS ITcoDoorLock
VAR_IN_OUT
    inoIsOpen : BOOL;
    inoIsLocked : BOOL;
    inoLock : BOOL;
END_VAR
VAR
    {attribute addProperty Name "<#Opened#>"}
    _isOpen : TcoElements.TcoDi(THIS^);

    {attribute addProperty Name "<#Locked#>"}
    _isLocked : TcoElements.TcoDi(THIS^);

    {attribute addProperty Name "<#Lock#>"}
    _lock : TcoElements.TcoDo(THIS^);


END_VAR

THIS^._isLocked(inoSignal :=  inoIsLocked);                    
THIS^._isOpen(inoSignal :=  inoIsOpen);                    
THIS^._lock(inoSignal   :=  inoLock);

PROPERTY IsClosed : BOOL
GET
IsClosed := THIS^._isOpen.IsFalse;
END_GET
END_PROPERTY

PROPERTY IsLocked : BOOL
GET
IsLocked := THIS^._isOpen.IsFalse and THIS^._isLocked.IsTrue ;
END_GET
END_PROPERTY

PROPERTY IsOpen : BOOL
GET
IsOpen := THIS^._isOpen.IsTrue;
END_GET
END_PROPERTY

METHOD Lock : BOOL
VAR_INPUT
END_VAR
Lock := FALSE;

THIS^._lock.Set();

IF	THIS^._isOpen.IsFalse THEN 
		
	IF THIS^._isLocked.IsTrue THEN 
		Lock := TRUE;
	END_IF
END_IF
END_METHOD

(*~
	<docu>
		<summary>
			Restores this instance to the Ready state. Can be called explicitly or from within one of the restore mechanisms.	
		</summary>			
	</docu>	
~*)
METHOD  Restore : ITcoRestorable
Unlock();
END_METHOD

(*~
	<docu>
		<summary>
		    Custom service (manual, maintenance) logic.
			This method must be implemented in derived class.
		</summary>			
	</docu>	
~*)
METHOD PROTECTED  ServiceMode
END_METHOD

METHOD UnLock : BOOL
VAR_INPUT
END_VAR

UnLock := FALSE;

THIS^._lock.Reset();
		
IF THIS^._isLocked.IsFalse THEN 
	UnLock := TRUE;
END_IF
END_METHOD

END_FUNCTION_BLOCK

// ---- Abstractions/Safety/Doors/TcoBasicDoor.TcPOU
FUNCTION_BLOCK TcoBasicDoor EXTENDS TcoCore.TcoComponent IMPLEMENTS ITcoDoorLock
VAR_IN_OUT
    inoIsClosed : BOOL;
    inoLock : BOOL;
END_VAR
VAR
    {attribute addProperty Name "<#Closed#>"}
    _isClosed : TcoElements.TcoDi(THIS^);

    {attribute addProperty Name "<#Lock#>"}
    _lock : TcoElements.TcoDo(THIS^);


END_VAR

                
THIS^._isClosed(inoSignal :=  inoIsClosed);                    
THIS^._lock(inoSignal   :=  inoLock);

PROPERTY IsClosed : BOOL
GET
IsClosed := THIS^._isClosed.IsTrue;
END_GET
END_PROPERTY

PROPERTY IsLocked : BOOL
GET
IsLocked := THIS^._isClosed.IsTrue and THIS^._lock.IsTrue ;
END_GET
END_PROPERTY

PROPERTY IsOpen : BOOL
GET
IsOpen := THIS^._isClosed.IsFalse;
END_GET
END_PROPERTY

METHOD Lock : BOOL
VAR_INPUT
END_VAR
Lock := FALSE;

THIS^._lock.Set();

IF	THIS^._isClosed.IsTrue THEN 
		Lock := TRUE;
END_IF
END_METHOD

(*~
	<docu>
		<summary>
			Restores this instance to the Ready state. Can be called explicitly or from within one of the restore mechanisms.	
		</summary>			
	</docu>	
~*)
METHOD  Restore : ITcoRestorable
UnLock();
END_METHOD

(*~
	<docu>
		<summary>
		    Custom service (manual, maintenance) logic.
			This method must be implemented in derived class.
		</summary>			
	</docu>	
~*)
METHOD PROTECTED  ServiceMode
END_METHOD

METHOD UnLock : BOOL
VAR_INPUT
END_VAR

UnLock := FALSE;

THIS^._lock.Reset();
		

UnLock := TRUE;
END_METHOD

END_FUNCTION_BLOCK

// ---- Abstractions/Safety/Estop/TcoEmergencyStop.TcPOU
{attribute wpf [Container(Layout.Stack)]}
FUNCTION_BLOCK TcoEmergencyStop EXTENDS TcoElements.TcoDi
VAR_OUTPUT
END_VAR
VAR
END_VAR

SUPER^(inoSignal:=inoSignal);
IF inoSignal THEN
	Messenger.Error('<#Emergency stop active#>').Pin();
END_IF;

END_FUNCTION_BLOCK

// ---- Abstractions/Safety/KeyMode/TcoKeyMode.TcPOU
{attribute wpf [Container(Layout.Stack)]}
FUNCTION_BLOCK TcoKeyMode EXTENDS TcoCore.TcoComponent IMPLEMENTS ITcoKeyMode
VAR_IN_OUT
	{attribute clr [RenderIgnore()]}
	inoKeyState1               : BOOL;
	
	{attribute clr [RenderIgnore()]}
	inoKeyState2               : BOOL;
END_VAR
VAR	
	
	{attribute addProperty Name "<#Status#>"}
    {attribute clr [ReadOnly()]}
    _status : TcoKeyMode_Status;

	{attribute addProperty Name "<#Config#>"}
    _config : TcoKeyMode_Config;
	{attribute addProperty Name "<#KeyState1#>"}
	KeyState1                : TcoElements.TcoDi(THIS^);
	
	{attribute addProperty Name "<#KeyState2#>"}
	KeyState2                : TcoElements.TcoDi(THIS^);
	
	//----------------- KEY STATES--------------
	{attribute addProperty Name "<#Manual#>"}
	IsKeyInManual            : BOOL; 
	
	{attribute addProperty Name "<#Automatic#>"}
	IsKeyInAuto              : BOOL; 
	
	{attribute addProperty Name "<#Step mode#>"}
	IsKeyInStep              : BOOL; 
	
	
	{attribute clr [RenderIgnore()]}
	_timer:ton;
END_VAR

KeyState1(inoSignal:= inoKeyState1);
KeyState2(inoSignal:= inoKeyState2);
_timer(IN:=(NOT KeyState1._signal   AND  KeyState2._signal) XOR (KeyState1._signal   AND  NOT KeyState2._signal),PT:=_config.SwitKeyStanilisiation);
THIS^.IsKeyInAuto   := KeyState1._signal       AND  KeyState2._signal;
THIS^.IsKeyInStep   := (NOT KeyState1._signal   AND  KeyState2._signal) XOR (KeyState1._signal   AND  NOT KeyState2._signal) AND _timer.Q;
THIS^.IsKeyInManual := NOT KeyState1._signal   AND  NOT KeyState2._signal;
//todo  timer

PROPERTY Config :REFERENCE TO TcoKeyMode_Config
GET
Config ref=_config;
END_GET
END_PROPERTY

PROPERTY KeyInAuto : BOOL
GET
KeyInAuto := IsKeyInAuto;
END_GET
END_PROPERTY

PROPERTY KeyInManual : BOOL
GET
KeyInManual := IsKeyInManual;
END_GET
END_PROPERTY

PROPERTY KeyInStep : BOOL
GET
KeyInStep := IsKeyInStep;
END_GET
END_PROPERTY

(*~
	<docu>
		<summary>
			Restores this instance to the Ready state. Can be called explicitly or from within one of the restore mechanisms.	
		</summary>			
	</docu>	
~*)
METHOD  Restore : ITcoRestorable
END_METHOD

(*~
	<docu>
		<summary>
		    Custom service (manual, maintenance) logic.
			This method must be implemented in derived class.
		</summary>			
	</docu>	
~*)
METHOD PROTECTED  ServiceMode
END_METHOD

PROPERTY Status : REFERENCE TO TcoKeyMode_Status
GET
Status REF=_status;
END_GET
END_PROPERTY

END_FUNCTION_BLOCK

// ---- Abstractions/Safety/KeyNormalService/TcoKeyNormalService.TcPOU
{attribute wpf [Container(Layout.Stack)]}
FUNCTION_BLOCK TcoKeyNormalService EXTENDS TcoElements.TcoDi IMPLEMENTS ITcoKeyNormalSevice

VAR

	
	{attribute addProperty Name "<#Key state#> - <#Service#>"}
	_isKeyInService           : BOOL; 

	{attribute addProperty Name "<#Key state#> - <#Normal#>"}
	_isKeyInNormal            : BOOL; 
END_VAR

SUPER^(inoSignal:= inoSignal);


THIS^._isKeyInNormal :=NOT THIS^._signal ;
THIS^._isKeyInService := NOT THIS^._isKeyInNormal;

PROPERTY KeyInNormal : BOOL
GET
KeyInNormal := _isKeyInNormal;
END_GET
END_PROPERTY

PROPERTY KeyInService : BOOL
GET
KeyInService := _isKeyInService;
END_GET
END_PROPERTY

END_FUNCTION_BLOCK
